INTERFACE ITF_BaseLoggerElement_HMI

END_INTERFACE

(* stored: Version 1.1.0.1
   Itf ITF_BaseLoggerElement_HMI: Id {5cb45a4d-d295-0879-1e7e-f79957b9c07c} *)
